Staubli VAL3: type.pgx

public program type(num x_nX, num x_nY, string x_sMessage)
begin
  //-----------------------------------------------------------------------
  //Header begin
  //Description of program
  //  Displays one string to pX column
  //  and pY Line.
  //
  //Input parameters
  //  num x_nX :
  //    role : Cursor column
  //  num x_nY :
  //    role : Cursor row
  //  string x_sMessage :
  //    role : Message that you want to display
  //
  //Example
  //  call type(2,5,"Staubli)
  //
  //History
  //  Creation : 28-04-08 - f.Rob
  //Header end
  //-----------------------------------------------------------------------
  gotoxy(x_nX,x_nY)
  put(x_sMessage)
end
